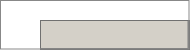
VISUALIZATION Ustawienia  // 190x50
    Button (40,20 150x30)
END_VISUALIZATION

(* stored: Version 1.1.0.1, ProductVersion 3.1.4024.11
   Visu Ustawienia: Id {b69ea445-69c9-45f8-a8c1-57da2a620837} *)
